(* PLC project op_chain, Dassault Systèmes ControlBuild 2024x *)
(* stored: creationDateTime 2023-10-03T11:13:59-01:00 *)

PROGRAM tri_chain.op_chain
  VAR_INPUT
    forward : BOOL := false;
  END_VAR
  VAR_OUTPUT
    localRun : BOOL := false;
    start_sensor : BOOL := false;
    end_sensor : BOOL := false;
  END_VAR

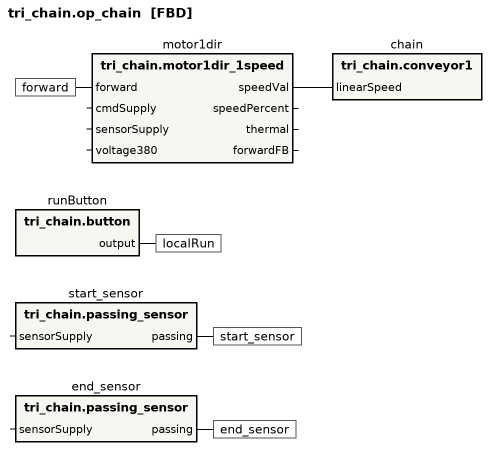
(* FBD diagram, written out as Structured Text *)
runButton();
localRun := runButton.output;
start_sensor();
start_sensor := start_sensor.passing;
end_sensor();
end_sensor := end_sensor.passing;
motor1dir(forward := forward);
chain(linearSpeed := motor1dir.speedVal);
END_PROGRAM
